INTERFACE I_CoeDevice EXTENDS I_Component, I_TaskResult

PROPERTY AdsAddr : REFERENCE TO AMSADDR
GET
END_GET
SET
END_SET
END_PROPERTY

METHOD Read
VAR_INPUT
	Index	 : WORD;
	SubIndex : BYTE;
	pDstBuf	 : PVOID;
	BufLen	 : UDINT;
END_VAR
END_METHOD

METHOD Write
VAR_INPUT
	Index	 : WORD;
	SubIndex : BYTE;
	pDstBuf	 : PVOID;
	BufLen	 : UDINT;
END_VAR
END_METHOD

END_INTERFACE

(* stored: Version 1.1.0.1, ProductVersion 3.1.4026.18
   Itf I_CoeDevice: Id {52ac7c54-bac3-4d07-a600-8b63f6b29713}
   Property AdsAddr: Id {e4aef1c7-deb0-4192-8a45-3c9cf80c2c77}
   Get Get: Id {609e8025-a4fe-4211-9dbd-0e6ff39c9ff1}
   Set Set: Id {269d1eb7-298b-43ec-a74f-e49be2af61bd}
   Method Read: Id {ed780fa2-4c1f-4680-ab7e-442d34f266f7}
   Method Write: Id {665c73f9-1118-465d-b85e-5662903bdff4} *)
